FUNCTION_BLOCK FB_Heatpump
VAR
	u_counter: UINT;
	InitSFC			:	FB_HeatPumpInit;
	OperationSFC	:	FB_HeatPumpOperation;
	
	//only written once at init.
	HeatPumpID		:	BYTE := 0;
END_VAR

VAR_STAT
	ui_Instancecounter : byte := 0;
END_VAR

VAR	
	MBMaster				: 	ModbusRtuMasterV2_KL6x22B;
	
	DataBuffer				:	ARRAY[0..50] OF WORD;
//	b_MBBusy				:	BOOL;
//	b_MBerr					:	BOOL;
//	ui_cbRead				:	UINT;
//	b_EnableTransmission	:	BOOL;
//	ModbusStartTrigger		:	R_Trig;
//	MBRetryCount			:	BYTE;
	
	
//	SendValue		:	WORD;
	
	OperatingPoint	:	st_OperatingPoint;
END_VAR

VAR_OUTPUT
	get			:	st_HeatpumpGet;
	MBCommBusy	:	BOOL := FALSE;
END_VAR

VAR_INPUT
	ACPowerStatus	:	BOOL;
	MBFree			:	BOOL;
END_VAR

//HeatpumpId is set once during first call
//var Stat InstanceCounter is shared between all functionblocks
IF HeatPumpId = 0 THEN
	ui_Instancecounter := ui_Instancecounter + 1;
	HeatPumpID := ui_Instancecounter ;
ELSE
	IF NOT ACPowerStatus THEN
		//Dont read all sensor data. Just monitor errors. We are not going to do anyting with the data anyway.
		InitSFC.SFCInit := TRUE;
		OperationSFC.SFCInit := TRUE;
		//OperationalSFC();
	ELSE
		InitSFC.SFCInit := FALSE;
		OperationSFC.SFCInit := FALSE;
	END_IF
END_IF

InitSFC(MBMaster := MBMaster, Get := Get, ACPowerSTatus := ACPowerStatus, HeatPumpID:=HeatPumpID);
OperationSFC(MBMaster := MBMaster, Get := Get, ACPowerSTatus := ACPowerStatus, HeatPumpID:=HeatPumpID,MBFree:=MBFree, OperatingPoint:=OperatingPoint, MBCommBusy=>MBCommbusy);

METHOD EMStop : BOOL
VAR_INPUT
END_VAR

get.HeatPumpState := eHeatpumpState.OFF;

EMstop := True;
END_METHOD

METHOD GetDiagnostics 
VAR_IN_OUT
	AddError		: ARRAY [*] OF FB_AddErrorST;
	a_ActiveEvents	: ARRAY [*] OF ST_ErrorStruct;
	w_Index			: WORD;
END_VAR

VAR_OUTPUT
	b_errorActive	: BOOL;
	b_warningActive	: BOOL;
END_VAR

VAR
	by_errCt	: BYTE;
	by_warnCt	: BYTE;
	w_ID		: WORD;
END_VAR
	(*Modbus comm fault*)	AddError[w_Index](
			in_b_ErrorTrig			:= Get.Events.b_CommError,
			out_ST_Error			:= a_ActiveEvents[w_Index],
			w_ID					:= 1 + w_ID,
			s_Message				:= 'Modbus communication error',
			e_sev					:= eSeverity.NormalShutdown,	
			in_b_AutoClear			:= FALSE,
			//in_e_ErrAckAccess		:= TRUE,
			);
		IF AddError[w_Index].b_out THEN by_errCt := by_errCt + 1; END_IF;
		w_Index := w_Index +1;
		
	(*Heatpump Compressor fault*)	AddError[w_Index](
			in_b_ErrorTrig			:= Get.Events.b_CompressorError,
			out_ST_Error			:= a_ActiveEvents[w_Index],
			w_ID					:= 2 + w_ID,
			s_Message				:= 'Heatpump Compressor fault',
			e_sev					:= eSeverity.NormalShutdown,	
			in_b_AutoClear			:= FALSE,
			//in_e_ErrAckAccess		:= TRUE,
			);
		IF AddError[w_Index].b_out THEN by_errCt := by_errCt + 1; END_IF;
		w_Index := w_Index +1;
	
	(*Heatpump Fan fault*)			AddError[w_Index](
			in_b_ErrorTrig			:= Get.Events.b_FanError,
			out_ST_Error			:= a_ActiveEvents[w_Index],
			w_ID					:= 3 + w_ID,
			s_Message				:= 'Heatpump Fan fault',
			e_sev					:= eSeverity.NormalShutdown,	
			in_b_AutoClear			:= FALSE,
			//in_e_ErrAckAccess		:= TRUE,
			);
		IF AddError[w_Index].b_out THEN by_errCt := by_errCt + 1; END_IF;
		w_Index := w_Index +1;
		
	(*HHeatpump Internal IO fault*)		AddError[w_Index](
			in_b_ErrorTrig			:= Get.Events.b_IOError ,
			out_ST_Error			:= a_ActiveEvents[w_Index],
			w_ID					:= 4 + w_ID,
			s_Message				:= 'Heatpump Internal IO fault',
			e_sev					:= eSeverity.NormalShutdown,	
			in_b_AutoClear			:= FALSE,
			//in_e_ErrAckAccess		:= TRUE,
			);
		IF AddError[w_Index].b_out THEN by_errCt := by_errCt + 1; END_IF;
		w_Index := w_Index +1;
		
	(*Heatpump pressure fault*)		AddError[w_Index](
			in_b_ErrorTrig			:= Get.Events.b_PressureError,
			out_ST_Error			:= a_ActiveEvents[w_Index],
			w_ID					:= 5 + w_ID,
			s_Message				:= 'Heatpump pressure fault',
			e_sev					:= eSeverity.NormalShutdown,	
			in_b_AutoClear			:= FALSE,
			//in_e_ErrAckAccess		:= TRUE,
			);
		IF AddError[w_Index].b_out THEN by_errCt := by_errCt + 1; END_IF;
		w_Index := w_Index +1;
		
	(*Heatpump Probe fault*)		AddError[w_Index](
			in_b_ErrorTrig			:= Get.Events.b_ProbeError,
			out_ST_Error			:= a_ActiveEvents[w_Index],
			w_ID					:= 6 + w_ID,
			s_Message				:= 'Heatpump Probe fault',
			e_sev					:= eSeverity.NormalShutdown,	
			in_b_AutoClear			:= FALSE,
			//in_e_ErrAckAccess		:= TRUE,
			);
		IF AddError[w_Index].b_out THEN by_errCt := by_errCt + 1; END_IF;
		w_Index := w_Index +1;	

	(*Heatpump Pump fault*)			AddError[w_Index](
			in_b_ErrorTrig			:= Get.Events.b_PumpError,
			out_ST_Error			:= a_ActiveEvents[w_Index],
			w_ID					:= 7 + w_ID,
			s_Message				:= 'Heatpump Pump fault',
			e_sev					:= eSeverity.NormalShutdown,	
			in_b_AutoClear			:= FALSE,
			//in_e_ErrAckAccess		:= TRUE,
			);
		IF AddError[w_Index].b_out THEN by_errCt := by_errCt + 1; END_IF;
		w_Index := w_Index +1;	

	(*Heatpump valve fault*)			AddError[w_Index](
			in_b_ErrorTrig			:= Get.Events.b_ValveError,
			out_ST_Error			:= a_ActiveEvents[w_Index],
			w_ID					:= 8 + w_ID,
			s_Message				:= 'Heatpump Valve fault',
			e_sev					:= eSeverity.NormalShutdown,	
			in_b_AutoClear			:= FALSE,
			//in_e_ErrAckAccess		:= TRUE,
			);
		IF AddError[w_Index].b_out THEN by_errCt := by_errCt + 1; END_IF;
		w_Index := w_Index +1;	

	(*Heatpump Water temperature error*)			AddError[w_Index](
			in_b_ErrorTrig			:= Get.Events.b_WaterTempError,
			out_ST_Error			:= a_ActiveEvents[w_Index],
			w_ID					:= 9 + w_ID,
			s_Message				:= 'Heatpump Water temperature error',
			e_sev					:= eSeverity.NormalShutdown,	
			in_b_AutoClear			:= FALSE,
			//in_e_ErrAckAccess		:= TRUE,
			);
		IF AddError[w_Index].b_out THEN by_errCt := by_errCt + 1; END_IF;
		w_Index := w_Index +1;	

(*Heatpump Comm warning*)			AddError[w_Index](
			in_b_ErrorTrig			:= Get.Events.b_commwarning,
			out_ST_Error			:= a_ActiveEvents[w_Index],
			w_ID					:= 10 + w_ID,
			s_Message				:= 'Heatpump communication warning',
			e_sev					:= eSeverity.Info,	
			in_b_AutoClear			:= TRUE,
			//in_e_ErrAckAccess		:= TRUE,
			);
		
		//for initial use, get notice if 1 packet fails. Clear immediately after datalogger run
		get.Events.b_CommWarning := FALSE;
END_METHOD

METHOD Reset : BOOL
VAR_INPUT
END_VAR
//until restarting the heatpump we don't know if errors are gone. So clear them for now.

get.Events.b_CommError := FALSE;
get.Events.b_CompressorError := FALSE;
get.Events.b_FanError := FALSE;
get.Events.b_IOError := FALSE;
get.Events.b_PressureError := FALSE;
get.Events.b_ProbeError := FALSE;
get.Events.b_PumpError := FALSE;
get.Events.b_ValveError := FALSE;
get.Events.b_WaterTempError := FALSE;

Reset := True;
END_METHOD

METHOD WriteSetpoint : BOOL
VAR_INPUT
	OperatingMode	:	eHeatpumpMode;
	SetPoint		: 	REAL;
END_VAR


OperatingPoint.OperatingMode := OperatingMode;
OperatingPoint.Setpoint := SetPoint;
END_METHOD

END_FUNCTION_BLOCK

(* stored: Version 1.1.0.1, ProductVersion 3.1.4024.12
   POU FB_Heatpump: Id {4d1361c4-7375-440c-8729-687ac25365b9}, SpecialFunc None
   Folder External methods: Id {ffbc8895-390e-4e55-bdb8-e7349cf6f2f6}
   Method EMStop: Id {5c418bf0-1070-4e41-8a2d-814833658cd1}
   Method getDiagnostics: Id {c255fa85-29b0-4377-b377-44c88c8da2f7}
   Method Reset: Id {1900faca-1d07-4824-9433-869147e176e5}
   Method WriteSetpoint: Id {4352f7d9-816c-47f1-a24b-96f628e791a8} *)
